FUNCTION_BLOCK Kitchen
VAR_INPUT
END_VAR
VAR_OUTPUT
END_VAR
VAR
END_VAR

END_FUNCTION_BLOCK

(* stored: Version 1.1.0.1, ProductVersion 3.1.4024.13
   POU Kitchen: Id {73ae86c2-6ef1-4252-ba9b-bc7850429b37}, SpecialFunc None *)
